{attribute 'qualified_only'}
{attribute 'strict'}
TYPE E_CustomErrorIds :
(
    //More information in: https://confluence.ess.eu/spaces/MCAG/pages/968065463/Custom+Error+IDs

    eNoCustomError := 0,
    eTemperatureSensorError := 16#10201,
    eAirPadPressureError := 16#10202,
    eExternalBrakeError := 16#10203,
    eExternalBrakeTimeoutError := 16#10204,
    eCommandHandlerTimeoutError := 16#10205
) UDINT := eNoCustomError;
END_TYPE
//  eTemperatureSensorError = '16#10201'
//  eAirPadPressureError = '16#10202'
//  eExternalBrakeError = '16#10203'
//  eExternalBrakeTimeoutError = '16#10204'
//  eCommandHandlerTimeoutError = '16#10205'

(* stored: Version 1.1.0.1
   EnumerationTextList E_CustomErrorIds: Id {12174a71-aafc-0e3e-2215-f2defb2a7324} *)
